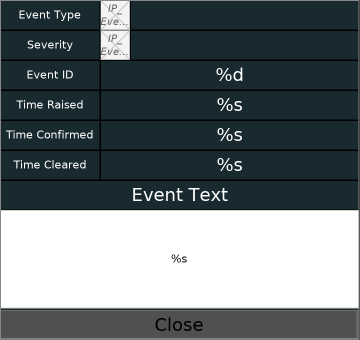
VISUALIZATION SingleEvent  // 360x340
VAR_IN_OUT
	data : ST_Event;
END_VAR
    Image (100,0 30x30), invisible if: data.iType <> 1, image: IP_EventType.alarm
    Image (100,0 30x30), invisible if: data.iType <> 2, image: IP_EventType.message
    Rectangle (130,0 230x30), text list: 'Event_Type', text index: data.iType
    Rectangle (0,0 100x30), "Event Type"
    Image (100,30 30x30), invisible if: data.eSeverity <> 4, image: IP_EventSeverity.critical
    Image (100,30 30x30), invisible if: data.eSeverity <> 3, image: IP_EventSeverity.error
    Image (100,30 30x30), invisible if: data.eSeverity <> 2, image: IP_EventSeverity.warning
    Image (100,30 30x30), invisible if: data.eSeverity <> 1, image: IP_EventSeverity.info
    Image (100,30 30x30), invisible if: data.eSeverity <> 0, image: IP_EventSeverity.verbose
    Rectangle (0,30 100x30), "Severity"
    Rectangle (130,30 230x30), text list: 'Event_Serverity', text index: data.eSeverity
    Rectangle (0,60 100x30), "Event ID"
    Rectangle (100,60 260x30), "%d", text variable: data.iEventId
    Rectangle (0,90 100x30), "Time Raised"
    Rectangle (100,90 260x30), "%s", text variable: LDT_TO_STRING(data.iTimeStamp)
    Rectangle (0,180 360x30), "Event Text"
    Textfield (-1,210 360x98), "%s", text variable: data.sEventText
    Button (-1,310 360x30), "Close"
        OnMouseClick: CloseDialog Dialog=SingleEvent, Result=Cancel, NumpadKeypadSet=True
    Rectangle (0,120 100x30), "Time Confirmed"
    Rectangle (100,120 260x30), "%s", text variable: LDT_TO_STRING(data.iTimeStampConfirmed)
    Rectangle (0,150 100x30), "Time Cleared"
    Rectangle (100,150 260x30), "%s", text variable: LDT_TO_STRING(data.iTimeStampCleared)
END_VISUALIZATION

(* stored: Version 1.1.0.1, ProductVersion 3.1.4024.9
   Visu SingleEvent: Id {7f4308a5-06c7-410a-aafd-8354e01a7f55} *)
